// SIMATIC S7-200 project (STEP 7-Micro/WIN), CPU 224XP REL 02.01

SYMBOL_TABLE USER1
start            I0.0     // start btn
stop_btn         I0.1     // stop btn
b1               I0.2     // bam 1
b2               I0.3     // bam 2
b3               I0.4     // bam 3
host             I0.5     // host
chuong           Q0.0     // chuong
d1               Q0.1     // den 1
d2               Q0.2     // den 2
d3               Q0.3     // den 3
END_SYMBOL_TABLE

ORGANIZATION_BLOCK MAIN:OB1
TITLE=PROGRAM COMMENTS
BEGIN
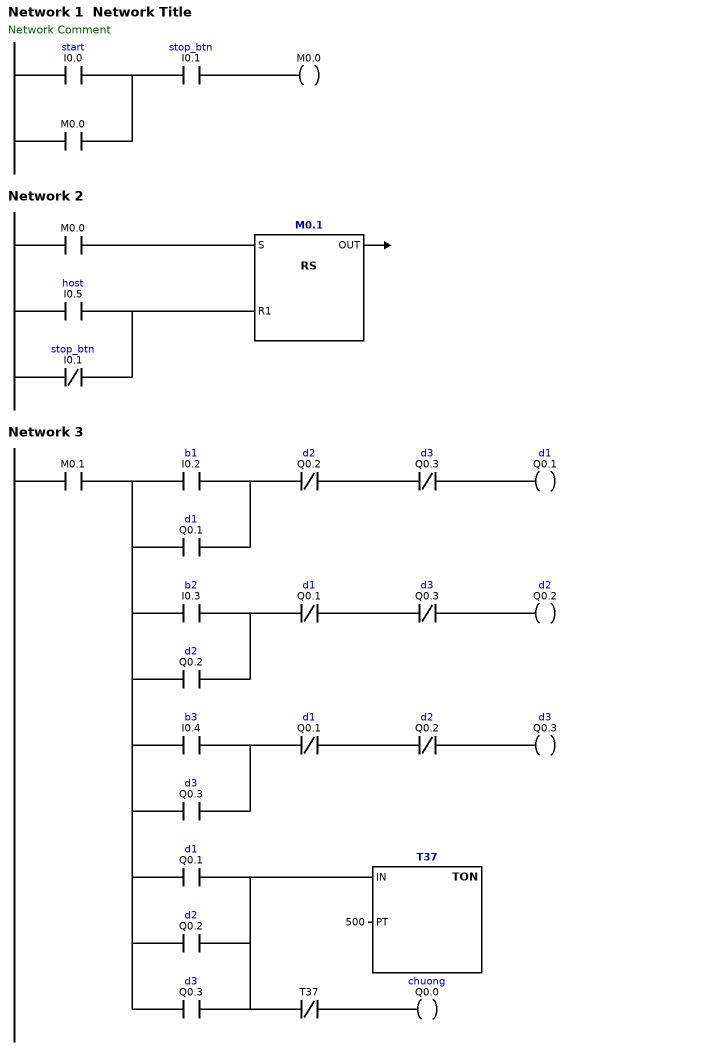
Network 1 // Network Title
// Network Comment
LD     start:I0.0
O      M0.0
A      stop_btn:I0.1
=      M0.0
Network 2
// (network saved uncompiled; LAD cells follow)
// row 0: c0 -| |- M0.0  c1 --  c2 [RS M0.1 S:=power@row0, R1:=power@row1, OUT=>power]  c3 ->
// row 1: c0 -| |- host:I0.5 v  c1 --  c2 [box]
// row 2: c0 -|/|- stop_btn:I0.1 ^
Network 3
// (network saved uncompiled; LAD cells follow)
// row 0: c0 -| |- M0.1 v  c1 -| |- b1:I0.2 v  c2 -|/|- d2:Q0.2  c3 -|/|- d3:Q0.3  c4 -( ) d1:Q0.1
// row 1: c0 ^v  c1 -| |- d1:Q0.1 ^
// row 2: c0 ^v  c1 -| |- b2:I0.3 v  c2 -|/|- d1:Q0.1  c3 -|/|- d3:Q0.3  c4 -( ) d2:Q0.2
// row 3: c0 ^v  c1 -| |- d2:Q0.2 ^
// row 4: c0 ^v  c1 -| |- b3:I0.4 v  c2 -|/|- d1:Q0.1  c3 -|/|- d2:Q0.2  c4 -( ) d3:Q0.3
// row 5: c0 ^v  c1 -| |- d3:Q0.3 ^
// row 6: c0 ^v  c1 -| |- d1:Q0.1 v  c2 --  c3 [TON T37 IN:=power@row6, PT:=500]
// row 7: c0 ^v  c1 -| |- d2:Q0.2 ^v  c3 [box]
// row 8: c0 ^  c1 -| |- d3:Q0.3 ^  c2 -|/|- T37  c3 -( ) chuong:Q0.0
END_ORGANIZATION_BLOCK
